KUKA KRL data list: KUKA_Server.dat

&ACCESS RVP
&REL 3
DEFDAT KUKA_SERVER PUBLIC

EXT BAS (BAS_COMMAND :IN, REAL :IN)
EXT KS_HANDLE_COMMAND(CHAR[] :IN)

DECL INT KS_RESULT
DECL INT KS_DEBUG_STEP
DECL INT KS_LAST_RECV_RESULT
DECL INT KS_LAST_SEND_RESULT
DECL INT KS_SEQUENCE
DECL INT KS_ACTIVE_SEQUENCE
DECL INT KS_BASE
DECL INT KS_TOOL

DECL CHAR KS_RX[2047]
DECL CHAR KS_LAST_RX[2047]
DECL CHAR KS_TX[2047]
DECL CHAR KS_MOTION_STATE[16]

DECL E6AXIS KS_AXIS_TARGET
DECL E6POS KS_POSE_TARGET

ENDDAT
